{attribute 'qualified_only'}
TYPE E_OpMod_ClsOpn :
(
	eClose			:= 0,
	eOpen			:= 1
	
) UDINT;
END_TYPE

(* stored: Version 1.1.0.1, ProductVersion 3.1.4024.5
   DUT E_OpMod_ClsOpn: Id {b9b32261-5ee4-40ec-9658-e1497a97e5c4} *)
